PROGRAM myBUTTONS
VAR
	rtHold: R_TRIG;
	bHoldCmd: bool;
	bRapidLed: BOOL;
END_VAR

PLCMachineMode[1].Start := bStartPB;
PLCMachineMode[1].Reset := bResetPB;

// Feedhold
bHoldLed := PLCMachineMode[0].ChannelSignals.FeedHold;
rtHold(CLK:= bHoldPB, Q=> );
IF rtHold.Q THEN
	bHoldCmd := NOT bHoldCmd;
END_IF
Global_HMI.PlcChannelSignals.FeedHold := bHoldCmd;

bRapidLed := stManualModeControlElements[0].stControlKeys[0].bKeyRapid;

PLCSpindleOverride := 50 + LREAL_TO_UINT(iSpindleOverridePot/32767.0*50.0); // limit overried to be 50% to 100?
IF PLCSpindleOverride > 99 THEN
	PLCSpindleOverride := 100;
ELSIF PLCSpindleOverride < 51 THEN
	PLCSpindleOverride := 50;
END_IF

PLCFeedOverride := 50 + LREAL_TO_UINT(iFeedrateOverridePot/32767.0*50.0); // limit overried to be 50% to 100?
IF PLCFeedOverride > 99 THEN
	PLCFeedOverride := 100;
ELSIF PLCFeedOverride < 51 THEN
	PLCFeedOverride := 50;
END_IF

END_PROGRAM

(* stored: Version 1.1.0.1, ProductVersion 3.1.4024.11
   POU myBUTTONS: Id {552323b9-8f8c-4a66-883f-ecc6de76eaee}, SpecialFunc None *)
